FUNCTION TryConvert_BYTE_TO_UINT : BOOL
VAR_INPUT
	in : BYTE;
	out : REFERENCE TO UINT;
END_VAR

out := BYTE_TO_UINT(in);
TryConvert_BYTE_TO_UINT := TRUE;

END_FUNCTION

(* stored: Version 1.1.0.1, ProductVersion 3.1.4024.12
   POU TryConvert_BYTE_TO_UINT: Id {31707e17-238e-4094-a545-b0fe15df55d7}, SpecialFunc None *)
